// Mitsubishi GX Works2 project: 10   PLC: FX3G

// task Task_01 (event TRUE, interval 0, priority 31): POU_01

PROGRAM POU_01
VAR
  wstep : INT;
  ton1 : TON;
  cnt : INT;
END_VAR
IF M8002 THEN
	wstep := 0;
	cnt := 0;
END_IF;

CASE wstep OF
	0:
		IF M0 THEN
			wstep := 20;
		END_IF;
		
	20:
		Z0 := cnt;
		Y0Z0 := TRUE;
		ton1(IN := NOT ton1.Q, PT := T#3s);
		IF ton1.Q THEN
			wstep := 21;
		END_IF;
	
	21:
		Y0Z0 := FALSE;
		cnt := cnt + 1;
		cnt := cnt MOD 3;
		
		wstep := 0;

END_CASE;
END_PROGRAM
